// Mitsubishi GX Works2 project: 智慧型停車塔-ST   PLC: FX3U/FX3UC
// 機電進階工業4.0智慧型停車塔物聯網控制系統

// task Task_01 (event TRUE, interval 0, priority 31): POU_01

PROGRAM POU_01
VAR
  wProgramStep : INT;
  bM1 : BOOL;
  tdTY6 : TON;
  tdT24 : TON;
  wC28 : INT;
  wPosNo : INT;
  arXZPos : ARRAY [0..23,0..1] OF INT;
  wC26 : INT;
  wC29 : INT;
  wC32 : INT;
  tdT23 : TON;
  tdT29 : TON;
  tdT32 : TON;
  wC30 : INT;
  bOut : BOOL;
  tdT41 : TON;
END_VAR
(* 機電整合智慧型停車塔
   實作部分: 自動入庫、出庫，手動入庫。
   Author: Steven Luo
   Date: 2018/09/26
*)

IF M8000 = TRUE THEN
	RS2(TRUE, D0, K0, K10, K1, D100);
END_IF;

IF M8002 AND X1 = TRUE THEN
	D8400 := H0C86; (* Baud rate: 9600, Data bits: 7, Parity check: Even, Stop bits: 1, RS-232 Normal 1 *)
	wProgramStep := 0;
	ZRST(TRUE, Y0, Y17);
	bM1 := FALSE;
END_IF;

IF M8403 = TRUE THEN
	RST(TRUE, M8403);
END_IF;

IF M8002 THEN
	wProgramStep := 21;
END_IF;

IF NOT X1 THEN (* 按下停止鈕 *)
	bM1 := TRUE;
END_IF;

IF NOT X2 AND X31 AND X24 AND NOT X36 THEN (* X軸馬達後退，Y軸滑台必須在正中 *)
	IF wProgramStep = 33 THEN
		tdT32(IN := FALSE);
		wProgramStep := 22;
	END_IF;
END_IF;

IF NOT X2 AND X16 THEN (* 入庫輸送 *)
	wProgramStep := 24;
END_IF;

IF NOT X2 AND X34 THEN (* Y軸馬達前進 *)
	IF wProgramStep = 24 THEN
		wProgramStep := 25;
	ELSIF wProgramStep = 30 THEN
		wProgramStep := 31;
	ELSIF wProgramStep = 32 THEN
		wProgramStep := 33;
	END_IF;
END_IF;

IF NOT X2 AND X32 THEN (* Z軸馬達上升 *)
	IF wProgramStep = 25 THEN
		wProgramStep := 26;
	ELSIF wProgramStep = 29 THEN
		wProgramStep := 30;
	END_IF;
END_IF;

IF NOT X2 AND X35 THEN (* Y軸馬達後退 *)
	IF wProgramStep = 26 THEN
		wProgramStep := 27;
	ELSIF wProgramStep = 30 THEN
		wProgramStep := 31;
	ELSIF wProgramStep = 32 THEN
		wProgramStep := 33;
	END_IF;
END_IF;

IF NOT X2 AND X30 THEN (* X軸馬達前進 *)
	IF wProgramStep = 28 THEN
		wProgramStep := 29;
	END_IF;
END_IF;

IF NOT X2 AND X33 THEN (* Z軸馬達下降 *)
	IF wProgramStep = 27 THEN
		wProgramStep := 28;
	ELSIF wProgramStep = 31 THEN
		wProgramStep := 32;
	END_IF;
END_IF;
(* 入庫動作: 22->23->24->25->26->27->28->29->30->31->32->33 *)
(* 出庫動作: 22->23->29->40->31->26->33->22->23->26->25->32->43 *)
CASE wProgramStep OF
	21:
		IF X1 (*AND X14 AND X24*) THEN (* 待機，按下啟動鈕 *)
			bM1 := FALSE;
			bOut := FALSE;
			FOR wPosNo := 0 TO 23 BY 1 DO
				IF wPosNo > 11 THEN
					arXZPos[wPosNo, 0] := (wPosNo - 12) / 3; (* X軸座標 0 ~ 3 *)
				ELSE
					arXZPos[wPosNo, 0] := wPosNo / 3; (* X軸座標 0 ~ 3 *)
				END_IF;
				arXZPos[wPosNo, 1] := (wPosNo MOD 3) + 1; (* Z軸座標 1 ~ 3 *)
			END_FOR;
		END_IF;
		IF X0 THEN
			wProgramStep := 22;
		END_IF;
	22: (* 回入庫原點 *)
		tdTY6(IN := FALSE);
		tdT24(IN := FALSE);
		tdT29(IN := FALSE);
		tdT32(IN := FALSE);
		tdT41(IN := FALSE);
		wC26 := 0;
		wC28 := 0;
		wC29 := 0;
		wC30 := 0;
		wC32 := 0;
		IF X24 AND NOT X36 THEN
			Y1 := TRUE;
		ELSE
			Y1 := FALSE;
		END_IF;
		IF NOT X24 THEN (* Y軸滑台移至正中 *)
			Y4 := TRUE;
			IF X26 THEN
				Y4 := FALSE;
				Y5 := TRUE;
			END_IF;
		ELSE
			IF Y4 THEN
				Y4 := FALSE;
			ELSE
				Y5 := FALSE;
			END_IF;
		END_IF;
		IF X24 AND NOT X37 THEN
			Y3 := TRUE;
		ELSE
			Y3 := FALSE;
		END_IF;
		IF X36 AND X24 AND X37 THEN
			Y0 := TRUE;
			tdT23(IN := FALSE);
 			wProgramStep := 23;
		END_IF;
	23:
		IF X14 THEN
			tdT23(IN := TRUE, PT := T#100ms);
			IF tdT23.Q THEN
				Y0 := FALSE;
				IF X2 THEN (* 自動 *)
					IF X3 THEN (* 出庫 *)
						IF bOut THEN
							wProgramStep := 26;
						ELSE
							D10 := K1X4;
							D11 := K1X10;
							wPosNo := D11 * 10 + D10 - 1;
							IF (wPosNo >= 0) OR (wPosNo <= 23) THEN
								wProgramStep := 28;
							END_IF;
						END_IF;
					ELSE (* 入庫 *)
						wProgramStep := 24;
			 		END_IF;
				END_IF;
			END_IF;
		END_IF;
	24:
		Y6 := TRUE; (* 入庫輸送 *)
		tdT24(IN := TRUE, PT := T#10s); (* 計時10秒 *)
		IF tdT24.Q THEN
			Y6 := FALSE;
			wProgramStep := 21;
		END_IF;
		IF X27 THEN (* 入庫輸送極限 *)
			tdTY6(IN := TRUE, PT := T#1s);
			IF tdTY6.Q THEN
				Y6 := FALSE;
				D10 := SHR(D100, K8);
				D11 := D100 AND H00FF;
				wPosNo := D10 - H30 + (D11 - H30) * 10 - 1;
				IF X2 THEN
					wProgramStep := 25;
				END_IF;
			END_IF;
		END_IF;
	25:
		Y4 := TRUE; (* Y軸滑台前進 *)
		IF X26 THEN
			Y4 := FALSE;
			IF X2 THEN
				IF X3 AND bOut THEN
					wProgramStep := 32;
				ELSE
					wProgramStep := 26;
				END_IF;
			END_IF;
		END_IF;
	26:
		Y2 := TRUE; (* Z軸馬達上升 *)
		INCP(X21, wC26);
		IF wC26 = 2 THEN
			Y2 := FALSE;
			IF X2 THEN
				IF X3 THEN
					IF bOut THEN
						wProgramStep := 25;
					ELSE
						wProgramStep := 33;
					END_IF;
				ELSE
					wProgramStep := 27;
				END_IF;
			END_IF;
		END_IF;
	27:
		Y5 := TRUE; (* Y軸滑台後退 *)
		IF X24 THEN (* 正中點 *)
			Y5 := FALSE;
			IF X2 THEN
				wProgramStep := 28;
			END_IF;
		END_IF;
	28:
		Y3 := TRUE; (* Z軸馬達下降 *)
		IF X37 THEN
			Y3 := FALSE;
			IF X2 THEN
				wProgramStep := 29;
			END_IF;
		END_IF;
	29:
		Y0 := TRUE; (* 移動至X座標 *)
		tdT29(IN := TRUE, PT := T#500ms);
		IF tdT29.Q THEN
			INCP(X14, wC29);
			IF wC29 > arXZPos[wPosNo, 0] THEN
				Y0 := FALSE;
				IF X2 THEN
					IF X3 THEN
						wProgramStep := 40;
					ELSE
						wProgramStep := 30;
					END_IF;
				END_IF;
			END_IF;
		END_IF;
	30:
		IF wC30 < (arXZPos[wPosNo, 1] * 2) THEN
			Y2 := TRUE; (* 移動至Z座標 *)
			INCP(X21, wC30);
		ELSE
			Y2 := FALSE;
			IF X2 THEN
				wProgramStep := 31;
			END_IF;
		END_IF;
	31:
		IF wPosNo < 12 THEN
			Y4 := TRUE; (* Y軸滑台前進 *)
			IF X26 THEN
				Y4 := FALSE;
				IF X2 THEN
					IF X3 THEN
						wProgramStep := 26;
					ELSE
						wProgramStep := 32;
					END_IF;
				END_IF;
			END_IF;
		ELSE
			Y5 := TRUE; (* Y軸滑台後退 *)
			IF X25 THEN
				Y5 := FALSE;
				IF X2 THEN
					IF X3 THEN
						wProgramStep := 26;
					ELSE
						wProgramStep := 32;
					END_IF;
				END_IF;
			END_IF;
		END_IF;
	32:
		Y3 := TRUE; (* Z軸馬達下降 *)
		tdT32(IN := TRUE, PT := T#3s);
		IF tdT32.Q THEN
			Y3 := FALSE;
			IF X2 THEN
				IF X3 AND bOut THEN
					wProgramStep := 43;
				ELSE
					wProgramStep := 33;
				END_IF;
			END_IF;
		END_IF;
	33:
		IF wPosNo < 12 THEN
			Y5 := TRUE; (* Y軸滑台後退 *)
			IF X24 THEN (* 正中點 *)
				Y5 := FALSE;
			END_IF;
		ELSE
			Y4 := TRUE; (* Y軸滑台前進 *)
			IF X24 THEN (* 正中點 *)
				Y4 := FALSE;
			END_IF;
		END_IF;
		IF X2 THEN
			IF X3 THEN
				bOut := TRUE;
			END_IF;
			wProgramStep := 22;
		END_IF;
	40:
		IF wC30 < (arXZPos[wPosNo, 1] * 2 - 1) THEN
			Y2 := TRUE; (* 移動至Z座標 *)
			INCP(X21, wC30);
		ELSE
			Y2 := FALSE;
			IF X2 THEN
				wProgramStep := 41;
			END_IF;
		END_IF;
	41:
		Y3 := TRUE;
		tdT41(IN := TRUE, PT := T#500ms);
		IF tdT41.Q THEN
			Y3 := FALSE;
			wProgramStep := 31;
		END_IF;
	43:
		Y7 := TRUE; (* 出庫輸送 *)
		tdT24(IN := TRUE, PT := T#3s); (* 計時3秒 *)
		IF tdT24.Q THEN
			Y7 := FALSE;
			wProgramStep := 21;
		END_IF;
	ELSE
	;
END_CASE;
END_PROGRAM
